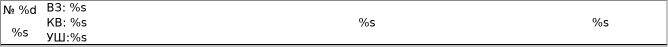
VISUALIZATION AlarmRecord_History_600  // 668x47
VAR_IN_OUT
	AlarmRecord: ST_AlarmRecord ; (*Запись об аварии для отображения*)
	RecNum: UINT; (*Номер записи*)
END_VAR
    Rectangle (196,0 342x45), "%s", text variable: AlarmRecord.Description
    Rectangle (40,0 154x15), "ВЗ: %s", text variable: AlarmRecord.Time_On
    Rectangle (40,15 154x15), "КВ: %s", text variable: AlarmRecord.Time_Quit
    Rectangle (40,30 155x15), "УШ:%s", text variable: AlarmRecord.Time_Off
    Rectangle (538,0 125x45), "%s", text variable: AlarmRecord.PossibleCause
    Rectangle (0,20 40x25), "%s", text variable: AlarmRecord.AlarmID, colour variable: AlarmRecord.Color
    Rectangle (0,0 40x20), "№ %d", text variable: RecNum
    Line (0,44) (666,44)
END_VISUALIZATION

(* stored: Version 1.1.0.1, ProductVersion 3.1.4024.2
   Visu AlarmRecord_History_600: Id {c033ab24-4836-44f7-92b0-416f9938a77f} *)
